(* PLC project op_door_locking, Dassault Systèmes ControlBuild 2024x *)
(* stored: creationDateTime 2023-10-03T11:13:50-01:00 *)

FUNCTION_BLOCK tni_train.op_door_locking
  VAR_INPUT
    lockingCmd : BOOL := false;
    unlockingCmd : BOOL := false;
  END_VAR
  VAR_OUTPUT
    doorLocked : BOOL := false;
    doorUnlocked : BOOL := false;
  END_VAR
  VAR_OUTPUT
    lockActive : BOOL := false;
  END_VAR
  VAR
    i_rs1 : DINT := 0;
  END_VAR
  VAR
    d_unlockedSensor : BOOL := false;
    v_d_unlockedSensor : BOOL := false;
    d_lockedSensor : BOOL := false;
    v_d_lockedSensor : BOOL := false;
  END_VAR

(* LD diagram, written out as Structured Text *)
1:
rs1(S := lockingCmd, R1 := unlockingCmd);
lockActive := rs1.Q1;
doorLocked := NOT d_lockedSensor AND lockActive OR d_lockedSensor AND v_d_lockedSensor;
doorUnlocked := NOT d_unlockedSensor AND NOT lockActive OR d_unlockedSensor AND v_d_unlockedSensor;
END_FUNCTION_BLOCK
